// TIA Portal project "Inversión de giro de motor temporizado" (V16)
// Implementación de la inversión de giro de un motor por meido de temporizadores, el motor inicia en un sentido tras pulsar incio, girará por un tiempo determinado, se detendrá por completo y empezará a girar en el otro sentido

(* hardware
DEVICE "S7-1200 station_1"  S7-1200 Station
   slot 0: "Rack_0"  S7-1200 Rack  Rack  V1.0
   slot 1: "PLC_1"  CPU 1214C DC/DC/DC  6ES7 214-1AG40-0XB0  V4.0
*)

// ===== PLC "PLC_1"  CPU 1214C DC/DC/DC =====

VAR_GLOBAL   // PLC tag table "Tabla de variables estándar"
   "START" AT %I0.0 : Bool;
   "STOP" AT %I0.1 : Bool;
   "T_Horario" AT %MD100 : Time;
   "T_Espera" AT %MD101 : Time;
   "T_Antihorario" AT %MD102 : Time;
   "M_Horario" AT %Q0.0 : Bool;
   "M_Antihorario" AT %Q0.1 : Bool;
   "Espera" AT %Q0.2 : Bool;
   "EsperaFinal" AT %Q0.3 : Bool;
   "T_Espera_Final" AT %MD103 : Time;
   "Final" AT %Q0.4 : Bool;
   "T_stop" AT %MD104 : Time;
   "Libre" AT %Q0.5 : Bool;
END_VAR

// folder: System blocks/Program resources

DATA_BLOCK "TemporizadorAntihorario"   // DB1
{ S7_Optimized_Access := 'TRUE' }
AUTHOR : Simatic
FAMILY : IEC
NAME : IEC_TMR
VERSION : 1.0
// stored: InstanceOfName IEC_TIMER
"IEC_TIMER"
BEGIN
END_DATA_BLOCK

DATA_BLOCK "TemporizadorEspera"   // DB2
{ S7_Optimized_Access := 'TRUE' }
AUTHOR : Simatic
FAMILY : IEC
NAME : IEC_TMR
VERSION : 1.0
// stored: InstanceOfName IEC_TIMER
"IEC_TIMER"
BEGIN
END_DATA_BLOCK

DATA_BLOCK "TemporizadorHorario"   // DB3
{ S7_Optimized_Access := 'TRUE' }
AUTHOR : Simatic
FAMILY : IEC
NAME : IEC_TMR
VERSION : 1.0
// stored: InstanceOfName IEC_TIMER
"IEC_TIMER"
BEGIN
END_DATA_BLOCK

DATA_BLOCK "TemporizadorEsperaFinal"   // DB4
{ S7_Optimized_Access := 'TRUE' }
AUTHOR : Simatic
FAMILY : IEC
NAME : IEC_TMR
VERSION : 1.0
// stored: InstanceOfName IEC_TIMER
"IEC_TIMER"
BEGIN
END_DATA_BLOCK

DATA_BLOCK "TemporizadorStop"   // DB5
{ S7_Optimized_Access := 'TRUE' }
AUTHOR : Simatic
FAMILY : IEC
NAME : IEC_TMR
VERSION : 1.0
// stored: InstanceOfName IEC_TIMER
"IEC_TIMER"
BEGIN
END_DATA_BLOCK

// folder: (top level)

ORGANIZATION_BLOCK "Main"   // OB1, LAD, ProgramCycle
TITLE = "Main Program Sweep (Cycle)" / Inversión de giro de motor temporizado
{ S7_Optimized_Access := 'TRUE' }
VERSION : 0.1
// Se arranca el motor en un sentido por un tiempo determinado, luego se detiene por un tiempo determinado, para arrancar en el otro sentido por un tiempo determinado, finalmente se detiene y espera un tiempo.
   VAR_INPUT
      Initial_Call : Bool;   // Initial call of this OB
      Remanence : Bool;   // =True, if remanent data are available
   END_VAR
BEGIN

REGION Network 1: Motor en sentido horario
   // Al pulsar "START" inicia el motor en sentido horario, se deshabilida o descativa cuando este en el proceso de espera de cambio de giro, cuando el motor esté girando en sentido antihorario, cuando este en la espera final, y cuando se haya pulsado "STOP", la varibale "Libre" es para espera un tiempo después de haber pulsado "STOP".
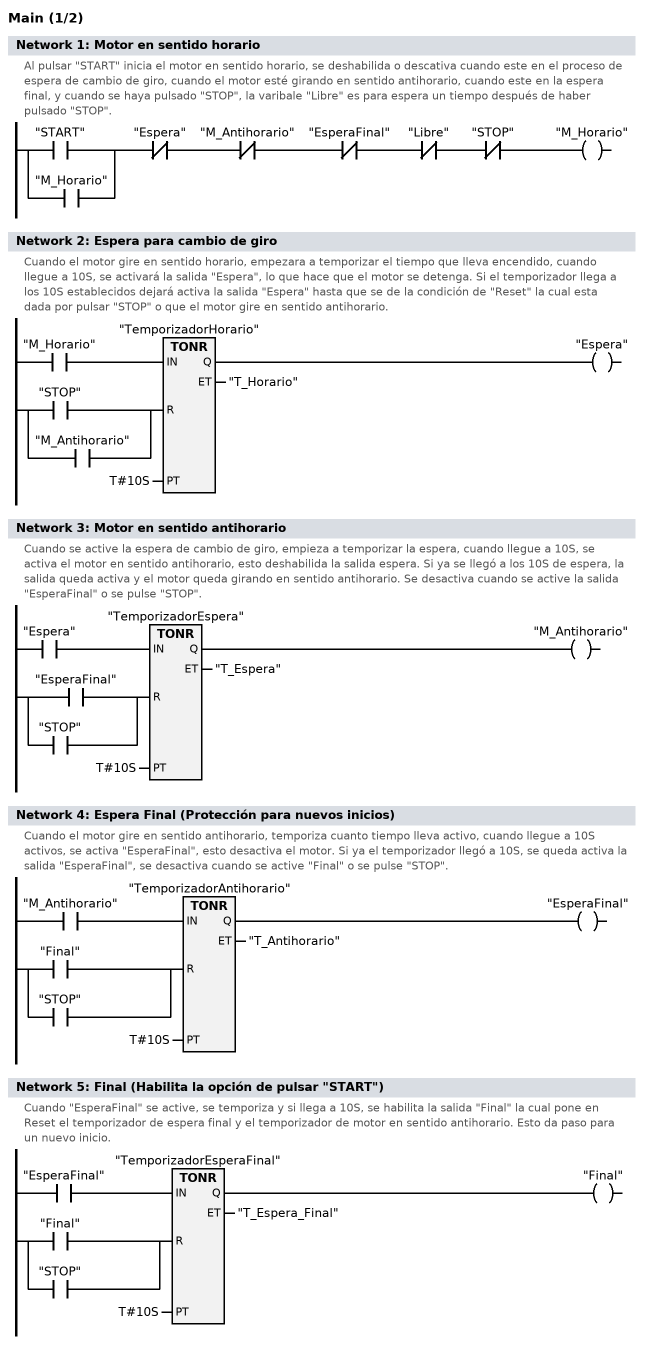
   RUNG wire#powerrail
      Contact( "START" )
      wire#w1
      I_Contact( "Espera" )
      I_Contact( "M_Antihorario" )
      I_Contact( "EsperaFinal" )
      I_Contact( "Libre" )
      I_Contact( "STOP" )
      Coil( "M_Horario" )
   END_RUNG
   RUNG wire#powerrail
      Contact( "M_Horario" )
   END_RUNG wire#w1
   // the same network as SCL:
   "M_Horario" := ("START" OR "M_Horario") AND NOT "Espera" AND NOT "M_Antihorario" AND NOT "EsperaFinal" AND NOT "Libre" AND NOT "STOP";
END_REGION

REGION Network 2: Espera para cambio de giro
   // Cuando el motor gire en sentido horario, empezara a temporizar el tiempo que lleva encendido, cuando llegue a 10S, se activará la salida "Espera", lo que hace que el motor se detenga. Si el temporizador llega a los 10S establecidos dejará activa la salida "Espera" hasta que se de la condición de "Reset" la cual esta dada por pulsar "STOP" o que el motor gire en sentido antihorario.
   "TemporizadorHorario".TONR(IN := "M_Horario", R := "STOP" OR "M_Antihorario", PT := T#10S, ET => "T_Horario");
   "Espera" := "TemporizadorHorario".Q;
END_REGION

REGION Network 3: Motor en sentido antihorario
   // Cuando se active la espera de cambio de giro, empieza a temporizar la espera, cuando llegue a 10S, se activa el motor en sentido antihorario, esto deshabilida la salida espera. Si ya se llegó a los 10S de espera, la salida queda activa y el motor queda girando en sentido antihorario. Se desactiva cuando se active la salida "EsperaFinal" o se pulse "STOP".
   "TemporizadorEspera".TONR(IN := "Espera", R := "EsperaFinal" OR "STOP", PT := T#10S, ET => "T_Espera");
   "M_Antihorario" := "TemporizadorEspera".Q;
END_REGION

REGION Network 4: Espera Final (Protección para nuevos inicios)
   // Cuando el motor gire en sentido antihorario, temporiza cuanto tiempo lleva activo, cuando llegue a 10S activos, se activa "EsperaFinal", esto desactiva el motor. Si ya el temporizador llegó a 10S, se queda activa la salida "EsperaFinal", se desactiva cuando se active "Final" o se pulse "STOP".
   "TemporizadorAntihorario".TONR(IN := "M_Antihorario",
                           R := "Final" OR "STOP",
                           PT := T#10S,
                           ET => "T_Antihorario");
   "EsperaFinal" := "TemporizadorAntihorario".Q;
END_REGION

REGION Network 5: Final (Habilita la opción de pulsar "START")
   // Cuando "EsperaFinal" se active, se temporiza y si llega a 10S, se habilita la salida "Final" la cual pone en Reset el temporizador de espera final y el temporizador de motor en sentido antihorario. Esto da paso para un nuevo inicio.
   "TemporizadorEsperaFinal".TONR(IN := "EsperaFinal",
                           R := "Final" OR "STOP",
                           PT := T#10S,
                           ET => "T_Espera_Final");
   "Final" := "TemporizadorEsperaFinal".Q;
END_REGION

REGION Network 6: Libre (Protección al pulsar "STOP")
   // Cuando se pulsa "STOP" se activa un temporizador de pulso, esto activa la salida "Libre" por 10S, esta salida deshabilida la condición de "START" haciendo que no sea posible iniciar inmediatamente después de pulsar "STOP".
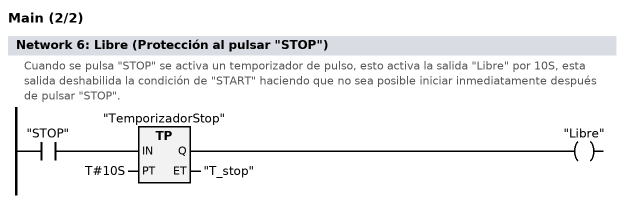
   "TemporizadorStop".TP(IN := "STOP", PT := T#10S, ET => "T_stop");
   "Libre" := "TemporizadorStop".Q;
END_REGION
END_ORGANIZATION_BLOCK